// TIA Portal V20 export
// export: Created 2026-07-14T14:10:11.1988747Z, ExportSetting WithDefaults, DisplayName Totally Integrated Automation Portal, DisplayVersion V20 Update 5, DisplayName TIA Portal Openness, DisplayVersion V20 Update 4, DisplayName TIA Portal Version Control Interface, DisplayVersion V20 Update 5, DisplayName SINAMICS Startdrive Advanced, DisplayVersion V20, DisplayName SINAMICS DCC, DisplayVersion V20, DisplayName SINAMICS Startdrive G130, G150, S120, S150, SINAMICS MV, G220, S200, S210, DisplayVersion V20, DisplayName SINAMICS Startdrive G110M, G120, G120C, G120D, G120P, G115D, DisplayVersion V20, DisplayName STEP 7 Professional, DisplayVersion V20 Update 5, DisplayName STEP 7 Safety, DisplayVersion V20 Update 2, DisplayName WinCC Basic/Comfort/Advanced, DisplayVersion V20 Update 5, DisplayName WinCC Unified, DisplayVersion V20 Update 5
FUNCTION "DataHandling" : Void   // FC22, LAD
{ S7_Optimized_Access := 'TRUE' }
VERSION : 0.1
// Data-handling reference examples (WAND/Calc/T_SUB/T_CONV/MOVE_BLK_VARIANT/Move)
// stored: AutoNumber true, IsIECCheckEnabled false, SetENOAutomatically false, UDAEnableTagReadback false
   VAR_TEMP
      DriveRunPermit : Bool;
      StatusWord : Word;
      DriveHealthy : Bool;
      DriveFaultReset : Bool;
      CommandWord : Word;
      Speed : Real;
      Ratio : Real;
      Divisor : Real;
      ScaledSpeed : Real;
      StartTime : Time;
      EndTime : Time;
      ElapsedTime : Time;
      ElapsedMillis : UDInt;
      SourceArray : Variant;
      ElementCount : UDInt;
      SourceStartIndex : UDInt;
      DestStartIndex : UDInt;
      MoveResult : Int;
      TargetArray : Variant;
      RunPermit : Bool;
      SourceValue : Int;
      StatusCode : Int;
   END_VAR
   VAR_TEMP   // added for the SCL form of the ladder/FBD networks
      _w1 : Bool;
   END_VAR
BEGIN

REGION Network 1: Drive command word (WAND)
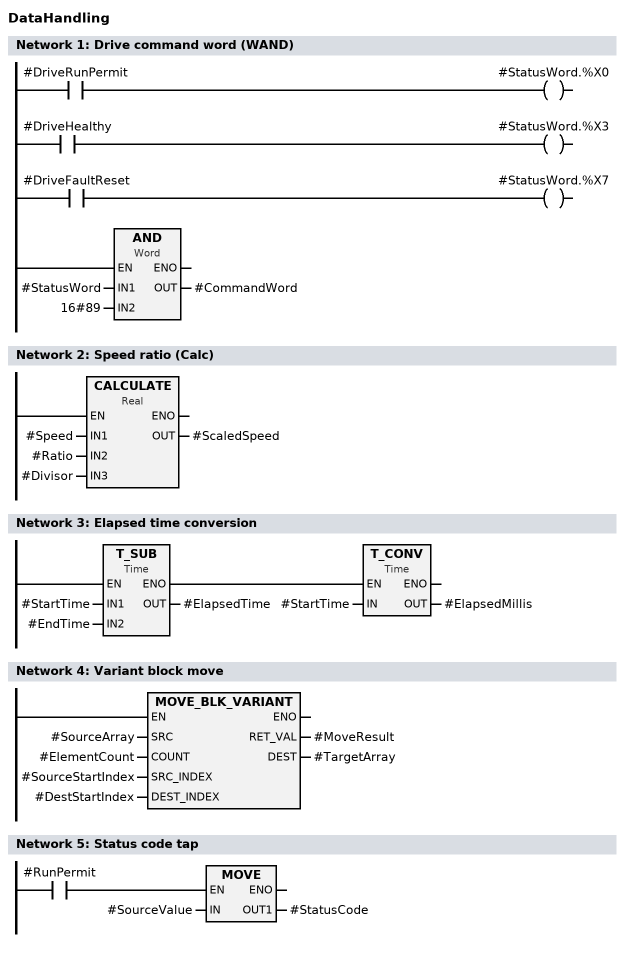
   RUNG wire#powerrail
      Contact( #DriveRunPermit )
      Coil( #StatusWord.%X0 )
   END_RUNG
   RUNG wire#powerrail
      Contact( #DriveHealthy )
      Coil( #StatusWord.%X3 )
   END_RUNG
   RUNG wire#powerrail
      Contact( #DriveFaultReset )
      Coil( #StatusWord.%X7 )
   END_RUNG
   RUNG wire#powerrail
      { S7_Templates := "SrcType := Word" } And(in1 := #StatusWord, in2 := 16#89, out => #CommandWord)
   END_RUNG
   // the same network as SCL:
   #StatusWord.%X0 := #DriveRunPermit;
   #StatusWord.%X3 := #DriveHealthy;
   #StatusWord.%X7 := #DriveFaultReset;
   #CommandWord := #StatusWord AND 16#89;
END_REGION

REGION Network 2: Speed ratio (Calc)
   RUNG wire#powerrail
      { S7_Templates := "SrcType := Real"; S7_Expression := "IN1*(IN2/IN3)" } Calculate(in1 := #Speed, in2 := #Ratio, in3 := #Divisor, out => #ScaledSpeed)
   END_RUNG
   // the same network as SCL:
   #ScaledSpeed := #Speed*(#Ratio/#Divisor);
END_REGION

REGION Network 3: Elapsed time conversion
   RUNG wire#powerrail
      { S7_Templates := "[date_type := Time, time_type := Time]" } T_SUB(IN1 := #StartTime, IN2 := #EndTime, OUT => #ElapsedTime)
      { S7_Templates := "[src_type := Time, dest_type := UDInt]" } T_CONV(IN := #StartTime, OUT => #ElapsedMillis)
   END_RUNG
   // the same network as SCL:
   T_SUB(IN1 := #StartTime, IN2 := #EndTime, OUT => #ElapsedTime, ENO => #_w1);
   IF #_w1 THEN T_CONV(IN := #StartTime, OUT => #ElapsedMillis); END_IF;
END_REGION

REGION Network 4: Variant block move
   RUNG wire#powerrail
      MOVE_BLK_VARIANT(SRC := #SourceArray, COUNT := #ElementCount, SRC_INDEX := #SourceStartIndex, DEST_INDEX := #DestStartIndex, Ret_Val => #MoveResult, DEST => #TargetArray)
   END_RUNG
   // the same network as SCL:
   #MoveResult := MOVE_BLK_VARIANT(SRC := #SourceArray,
                           COUNT := #ElementCount,
                           SRC_INDEX := #SourceStartIndex,
                           DEST_INDEX := #DestStartIndex,
                           DEST => #TargetArray);
END_REGION

REGION Network 5: Status code tap
   RUNG wire#powerrail
      Contact( #RunPermit )
      Move(in := #SourceValue, out1 => #StatusCode)
   END_RUNG
   // the same network as SCL:
   IF #RunPermit THEN #StatusCode := #SourceValue; END_IF;
END_REGION
END_FUNCTION
